Omron CX-Programmer project NewProject (CX-Programmer 9.72)

# PLC NodeA: CP2E-N N

## Global symbols (name address type ; comment)
D9000 CHANNEL  ; Send_NodeB_ErrorCode
D9001 CHANNEL  ; Receive_NodeB_Errorcode
D9002 CHANNEL  ; Send_NodeC_ErrorCode
D9003 CHANNEL  ; Receive_NodeC_ErrorCode
D9004 CHANNEL  ; Send_NodeD_ErrorCode
D9005 CHANNEL  ; Receive_NodeD_ErrorCode
W10.00 BOOL  ; Send_NodeB
W10.01 BOOL  ; Send_NodeB_BUSY
W10.02 BOOL  ; Send_NodeB_OK
W10.03 BOOL  ; Send_NodeB_NG
W11.00 BOOL  ; Receive_NodeB
W11.01 BOOL  ; Receive_NodeB_BUSY
W11.02 BOOL  ; Receive_NodeB_OK
W11.03 BOOL  ; Receive_NodeB_NG
W12.00 BOOL  ; Send_NodeC
W12.01 BOOL  ; Send_NodeC_BUSY
W12.02 BOOL  ; Send_NodeC_OK
W12.03 BOOL  ; Send_NodeC_NG
W13.00 BOOL  ; Receive_NodeC
W13.01 BOOL  ; Receive_NodeC BUSY
W13.02 BOOL  ; Receive_NodeC_OK
W13.03 BOOL  ; Receive_NodeC_NG
W14.00 BOOL  ; Send_NodeD
W14.01 BOOL  ; Send_NodeD_BUSY
W14.02 BOOL  ; Send_NodeD_OK
W14.03 BOOL  ; Send_NodeD_NG
W15.00 BOOL  ; Receive_NodeD
W15.01 BOOL  ; Receive_NodeD_BUSY
W15.02 BOOL  ; Receive_NodeD_OK
W15.03 BOOL  ; Receive_NodeD_NG
Receive_NodeB _CPxx002_ReceiveData
Receive_NodeC _CPxx002_ReceiveData
Receive_NodeD _CPxx002_ReceiveData
Send_NodeB _CPxx001_SendData
Send_NodeC _CPxx001_SendData
Send_NodeD _CPxx001_SendData

## Program NewProgram1 (cyclic task 0)

### Section Section1

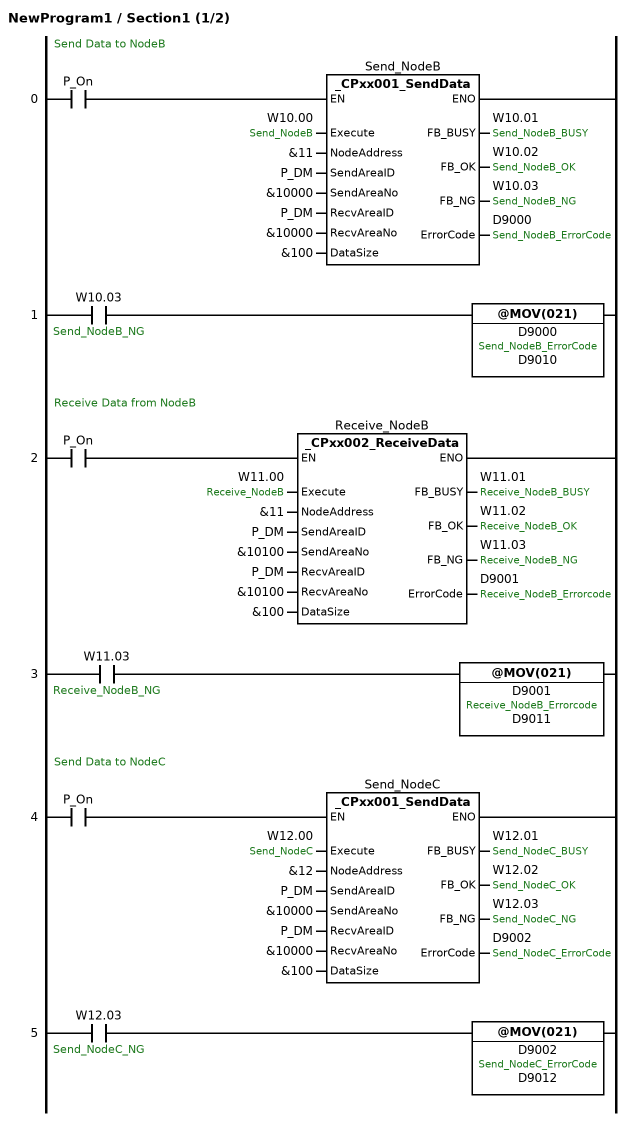
; rung 0: Send Data to NodeB
LD P_On
CALL Send_NodeB : _CPxx001_SendData (Execute := W10.00, NodeAddress := &11, SendAreaID := P_DM, SendAreaNo := &10000, RecvAreaID := P_DM, RecvAreaNo := &10000, DataSize := &100, FB_BUSY => W10.01, FB_OK => W10.02, FB_NG => W10.03, ErrorCode => D9000)  ; Send_NodeB, Send_NodeB_BUSY, Send_NodeB_OK, Send_NodeB_NG, Send_NodeB_ErrorCode
; rung 1
LD W10.03  ; Send_NodeB_NG
@MOV(021) D9000 D9010  ; Send_NodeB_ErrorCode
; rung 2: Receive Data from NodeB
LD P_On
CALL Receive_NodeB : _CPxx002_ReceiveData (Execute := W11.00, NodeAddress := &11, SendAreaID := P_DM, SendAreaNo := &10100, RecvAreaID := P_DM, RecvAreaNo := &10100, DataSize := &100, FB_BUSY => W11.01, FB_OK => W11.02, FB_NG => W11.03, ErrorCode => D9001)  ; Receive_NodeB, Receive_NodeB_BUSY, Receive_NodeB_OK, Receive_NodeB_NG, Receive_NodeB_Errorcode
; rung 3
LD W11.03  ; Receive_NodeB_NG
@MOV(021) D9001 D9011  ; Receive_NodeB_Errorcode
; rung 4: Send Data to NodeC
LD P_On
CALL Send_NodeC : _CPxx001_SendData (Execute := W12.00, NodeAddress := &12, SendAreaID := P_DM, SendAreaNo := &10000, RecvAreaID := P_DM, RecvAreaNo := &10000, DataSize := &100, FB_BUSY => W12.01, FB_OK => W12.02, FB_NG => W12.03, ErrorCode => D9002)  ; Send_NodeC, Send_NodeC_BUSY, Send_NodeC_OK, Send_NodeC_NG, Send_NodeC_ErrorCode
; rung 5
LD W12.03  ; Send_NodeC_NG
@MOV(021) D9002 D9012  ; Send_NodeC_ErrorCode

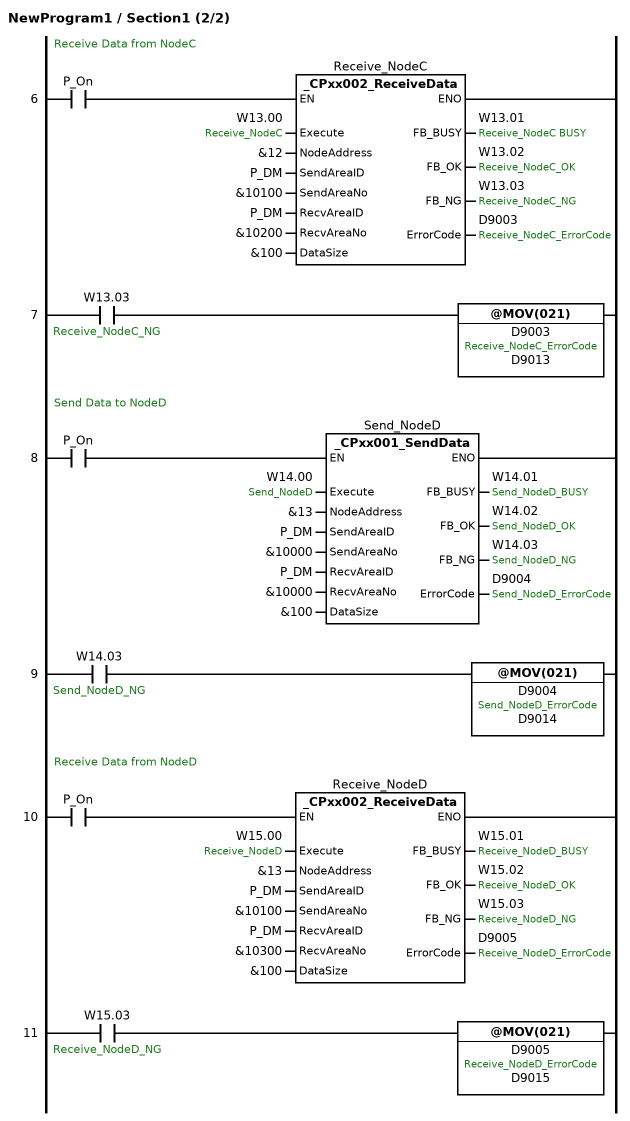
; rung 6: Receive Data from NodeC
LD P_On
CALL Receive_NodeC : _CPxx002_ReceiveData (Execute := W13.00, NodeAddress := &12, SendAreaID := P_DM, SendAreaNo := &10100, RecvAreaID := P_DM, RecvAreaNo := &10200, DataSize := &100, FB_BUSY => W13.01, FB_OK => W13.02, FB_NG => W13.03, ErrorCode => D9003)  ; Receive_NodeC, Receive_NodeC BUSY, Receive_NodeC_OK, Receive_NodeC_NG, Receive_NodeC_ErrorCode
; rung 7
LD W13.03  ; Receive_NodeC_NG
@MOV(021) D9003 D9013  ; Receive_NodeC_ErrorCode
; rung 8: Send Data to NodeD
LD P_On
CALL Send_NodeD : _CPxx001_SendData (Execute := W14.00, NodeAddress := &13, SendAreaID := P_DM, SendAreaNo := &10000, RecvAreaID := P_DM, RecvAreaNo := &10000, DataSize := &100, FB_BUSY => W14.01, FB_OK => W14.02, FB_NG => W14.03, ErrorCode => D9004)  ; Send_NodeD, Send_NodeD_BUSY, Send_NodeD_OK, Send_NodeD_NG, Send_NodeD_ErrorCode
; rung 9
LD W14.03  ; Send_NodeD_NG
@MOV(021) D9004 D9014  ; Send_NodeD_ErrorCode
; rung 10: Receive Data from NodeD
LD P_On
CALL Receive_NodeD : _CPxx002_ReceiveData (Execute := W15.00, NodeAddress := &13, SendAreaID := P_DM, SendAreaNo := &10100, RecvAreaID := P_DM, RecvAreaNo := &10300, DataSize := &100, FB_BUSY => W15.01, FB_OK => W15.02, FB_NG => W15.03, ErrorCode => D9005)  ; Receive_NodeD, Receive_NodeD_BUSY, Receive_NodeD_OK, Receive_NodeD_NG, Receive_NodeD_ErrorCode
; rung 11
LD W15.03  ; Receive_NodeD_NG
@MOV(021) D9005 D9015  ; Receive_NodeD_ErrorCode

### Section END
; rung 0
END(001)

## Function block _CPxx001_SendData (Omron library block, body left out)

## Function block _CPxx002_ReceiveData (Omron library block, body left out)

# PLC NodeB: CP2E-N N

## Program NewProgram1 (cyclic task 0)

### Section Section1

### Section END
; rung 0
END(001)

# PLC NodeC: CP2E-N N

## Program NewProgram1 (cyclic task 0)

### Section Section1

### Section END
; rung 0
END(001)

# PLC NodeD: CP2E-N N

## Program NewProgram1 (cyclic task 0)

### Section Section1

### Section END
; rung 0
END(001)